FUNCTION_BLOCK SS4_ps_Laser (* Composite FB wrapping other FBs *)
  (* Standard: 61499-2 *)
  (* Version 1.0, 2025-08-25, PS_Transformer_for_Unknown *)
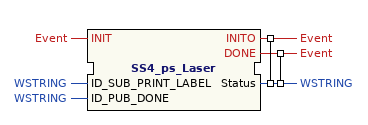
  EVENT_INPUT
    INIT; (* Initialization Request *)
  END_EVENT
  EVENT_OUTPUT
    INITO WITH Status; (* Initialization Confirm *)
    DONE WITH Status; (* Execution Confirmation *)
  END_EVENT
  VAR_INPUT
    ID_SUB_PRINT_LABEL : WSTRING;
    ID_PUB_DONE : WSTRING;
  END_VAR
  VAR_OUTPUT
    Status : WSTRING; (* Output event qualifier *)
  END_VAR
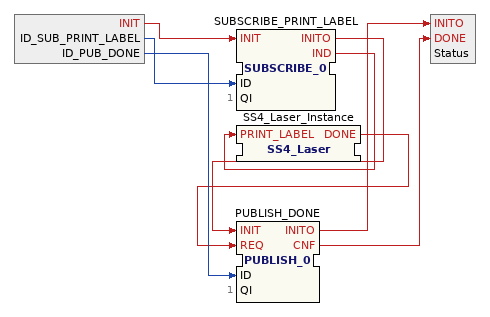
  FBS
    SS4_Laser_Instance : SS4_Laser;
    SUBSCRIBE_PRINT_LABEL : SUBSCRIBE_0(QI := 1);
    PUBLISH_DONE : PUBLISH_0(QI := 1);
  END_FBS
  EVENT_CONNECTIONS
    INIT TO SUBSCRIBE_PRINT_LABEL.INIT;
    SUBSCRIBE_PRINT_LABEL.INITO TO PUBLISH_DONE.INIT;
    PUBLISH_DONE.INITO TO INITO;
    SUBSCRIBE_PRINT_LABEL.IND TO SS4_Laser_Instance.PRINT_LABEL;
    SS4_Laser_Instance.DONE TO PUBLISH_DONE.REQ;
    PUBLISH_DONE.CNF TO DONE;
  END_CONNECTIONS
  DATA_CONNECTIONS
    ID_SUB_PRINT_LABEL TO SUBSCRIBE_PRINT_LABEL.ID;
    ID_PUB_DONE TO PUBLISH_DONE.ID;
  END_CONNECTIONS
END_FUNCTION_BLOCK
